TYPE DUT_Com_Base_Valve :
STRUCT
	Open :BOOL;
	Close :BOOL;
	Reset :BOOL;
	Simulation :BOOL;
	AutoOn :BOOL;
	AutoOff :BOOL;
	ManualOn :BOOL;
	ManualOff :BOOL;
END_STRUCT
END_TYPE

(* stored: Version 1.1.0.1, ProductVersion 3.1.4024.12
   DUT DUT_Com_Base_Valve: Id {b6e1d523-0f0a-41db-aa44-7681e860b370} *)
